FUNCTION_BLOCK MachineSequenceGoHome EXTENDS MachineSequence IMPLEMENTS ZCore.ISequence
VAR
  _step : ZCore.Step(MachineStep.GohomeBegin, MachineStep.GohomeEnd);
  _timer : ZAux.Timer;
END_VAR

IF NOT Busy THEN
  RETURN;
END_IF

IF OnStart(_step) THEN
  ; // init custom sequence variables here ...
END_IF

IF OnStop() THEN
  RETURN; // external stop was triggered
END_IF

IF OnHalt() THEN
  ; // Halting := TRUE; // Uncomment to acknowledge that the sequence is halting
END_IF

REPEAT
  LogStep();

  CASE _step.Index OF
    (* -------------------------------------------------------------------------------------------------------------------------------- *)
    MachineStep.GoHomeBegin:
    (* -------------------------------------------------------------------------------------------------------------------------------- *)
      IF _step.OnEntry()
      THEN
        _axis.ToolX.MoveAbsoluteAsync(THIS^, 300, _data.Machine.Slowspeed);
        _axis.TransportX.HomingAsync(THIS^);  
			END_IF
      
      Await2(_axis.ToolX, _axis.TransportX, nextStep:=MachineStep.GoHomeEnd);

    (* -------------------------------------------------------------------------------------------------------------------------------- *)
    MachineStep.GoHomeEnd:
    (* -------------------------------------------------------------------------------------------------------------------------------- *)
      SetBusy(FALSE);
  
  ELSE
    Abort('sequence contains unhandled step');
  END_CASE
UNTIL _step.IsNotRepeatable() OR_ELSE NOT Busy END_REPEAT

END_FUNCTION_BLOCK

(* stored: Version 1.1.0.1
   POU MachineSequenceGoHome: Id {2a1b1cde-3c5c-4242-b6c6-d89042e3e2c8}, SpecialFunc None *)
